# EPICS autosave request: BPMRFFEApp/Db/BPMRFFE_settings.req
file "BPMRffe_settings.req",   P=$(P)
